// How to initialize plant control with helper methods in "FB_init()".
// [Hint]
// > All reference-variables are implemented to ease monitoring of relevant variables.
FUNCTION_BLOCK FB_Plt_Init2 EXTENDS FB_BA_View
VAR
   	{region 'Aggregates'}
		DmprSu_Open							: REFERENCE TO BOOL							REF= DmprSu.bOpen;
		DmprSu_Val							: REFERENCE TO REAL							REF= DmprSu.fActiveVal;
		DmprSu								: FB_TimerAggregateA						:= (iParent:=THIS^,					iLabel:=MyLabels.DmprSu);
		FanSu_Val							: REFERENCE TO UDINT						REF= FanSu.nActiveVal;
		FanSu								: FB_BA_AggregateM							:= (iParent:=THIS^,					iLabel:=MyLabels.FanSu);
			 
		DmprEx_Open							: REFERENCE TO BOOL							REF= DmprEx.bOpen;
		DmprEx_Val							: REFERENCE TO REAL							REF= DmprEx.fActiveVal;
		DmprEx								: FB_TimerAggregateA						:= (iParent:=THIS^,					iLabel:=MyLabels.DmprEx);
		FanEx_Val							: REFERENCE TO UDINT						REF= FanEx.nActiveVal;
		FanEx								: FB_BA_AggregateM							:= (iParent:=THIS^,					iLabel:=MyLabels.FanEx);
			 
		PreHtr_Proc							: REFERENCE TO BOOL							REF= PreHtr.Process.bActive;
		PreHtr_Val							: REFERENCE TO BOOL							REF= PreHtr.bActiveVal;
		PreHtr								: FB_ProcAggregateB							:= (iParent:=THIS^,					iLabel:=MyLabels.PreHtr,			Process:=(iLabel:=MyLabels.ProcPreRinse));
		Erc_Val								: REFERENCE TO BOOL							REF= Erc.bActiveVal;
		Erc									: FB_BA_AggregateB							:= (iParent:=THIS^,					iLabel:=MyLabels.Erc);
		Col_Val								: REFERENCE TO BOOL							REF= Col.bActiveVal;
		Col									: FB_BA_AggregateB							:= (iParent:=THIS^,					iLabel:=MyLabels.Col);
	{endregion}
	{region 'Plant'} 
		OpMode								: E_OpMod_AC								:= E_OpMod_AC.eOff;
		PlantCtrl_OpSta						: REFERENCE TO BOOL							REF= PlantCtrl.bOpSta;
		PlantCtrl_On						: REFERENCE TO BOOL							REF= PlantCtrl.bOn;
		PlantCtrl_PrVal						: REFERENCE TO UDINT						REF= PlantCtrl.nPresentValue;
		PlantCtrl_Step						: REFERENCE TO STRING						REF= PlantCtrl.sStep;
		PlantCtrl							: FB_BA_PlantCtrl							:= (iParent:=THIS^,					iLabel:=MyLabels.PltCtrl);
	{endregion}
END_VAR

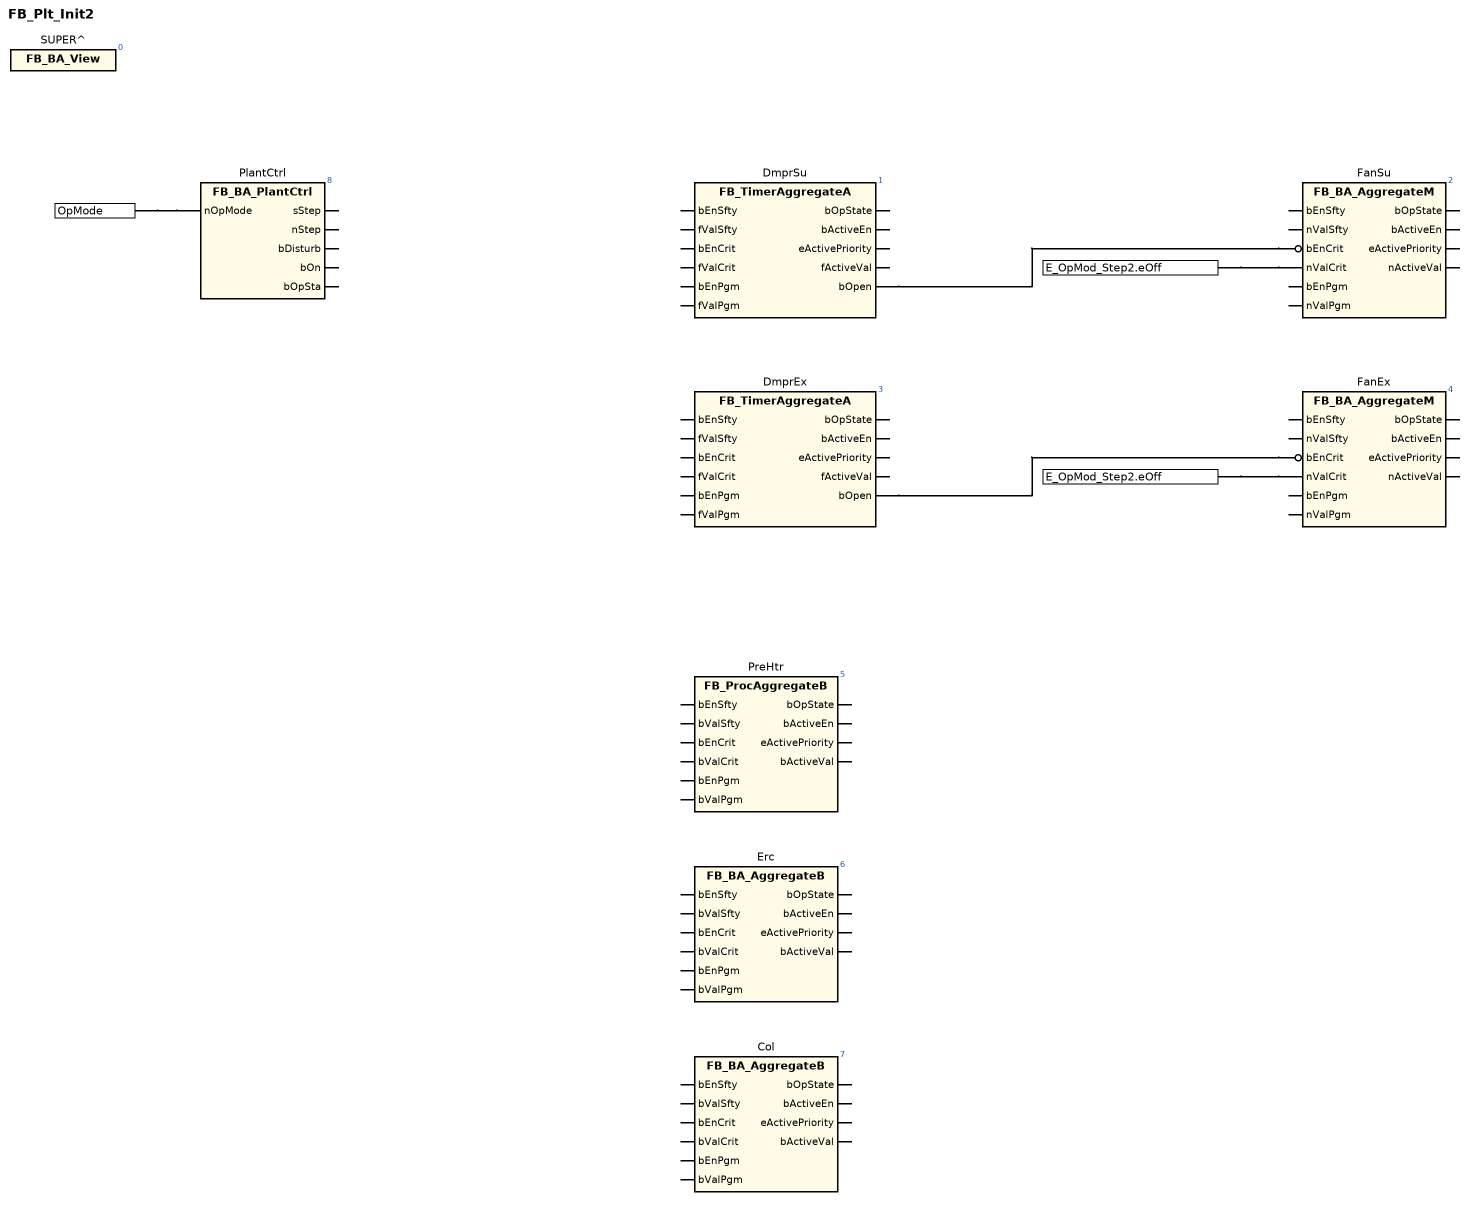
SUPER^(); // FB_BA_View
DmprSu(); // FB_TimerAggregateA
FanSu(bEnCrit := NOT DmprSu.bOpen, nValCrit := E_OpMod_Step2.eOff); // FB_BA_AggregateM
DmprEx(); // FB_TimerAggregateA
FanEx(bEnCrit := NOT DmprEx.bOpen, nValCrit := E_OpMod_Step2.eOff); // FB_BA_AggregateM
PreHtr(); // FB_ProcAggregateB
Erc(); // FB_BA_AggregateB
Col(); // FB_BA_AggregateB
PlantCtrl(nOpMode := OpMode); // FB_BA_PlantCtrl

METHOD FB_init : BOOL
VAR_INPUT
	bInitRetains : BOOL; // if TRUE, the retain variables are initialized (warm start / cold start)
	bInCopyCode : BOOL;  // if TRUE, the instance afterwards gets moved into the copy code (online change)
END_VAR
PlantCtrl.Clear();

// Add plant operations modes:
PlantCtrl.AddOperationMode(E_OpMod_AC.eDisturb,			E_BA_Priority.eCritical,	E_BA_AggregateIgnoreFlags.Delay);
PlantCtrl.AddOperationMode(E_OpMod_AC.eSmokeExtract,	E_BA_Priority.eLifeSafety,	E_BA_AggregateIgnoreFlags.All);
PlantCtrl.AddOperationMode(E_OpMod_AC.eOff,				E_BA_Priority.eProgram,		E_BA_AggregateIgnoreFlags.None);
PlantCtrl.AddOperationMode(E_OpMod_AC.eOn,				E_BA_Priority.eProgram,		E_BA_AggregateIgnoreFlags.None);
PlantCtrl.AddOperationMode(E_OpMod_AC.eNightCool,		E_BA_Priority.eProgram,		E_BA_AggregateIgnoreFlags.None);

// Add aggregates:
PlantCtrl.AddAggregate(DmprSu,	FALSE,	FALSE,	T#0S,	T#0S);
PlantCtrl.AddAggregate(DmprEx,	FALSE,	FALSE,	T#0S,	T#0S);
PlantCtrl.AddAggregate(PreHtr,	TRUE,	FALSE,	T#0S,	T#0S);
PlantCtrl.AddAggregate(Erc,		FALSE,	FALSE,	T#0S,	T#0S);
PlantCtrl.AddAggregate(Col,		FALSE,	FALSE,	T#0S,	T#0S);
PlantCtrl.AddAggregate(FanSu,	FALSE,	FALSE,	T#0S,	T#5S);
PlantCtrl.AddAggregate(FanEx,	FALSE,	FALSE,	T#5S,	T#0S);

// Apply aggregate operation modes dependant on corresponding plant operation modes:
PlantCtrl.AssignAggregate4x(E_OpMod_AC.eDisturb,		DmprSu, TO_UDINT(0),					FanSu, TO_UDINT(E_OpMod_Step2.eOff),		DmprEx, TO_UDINT(0),					FanEx, TO_UDINT(E_OpMod_Step2.eOff));
PlantCtrl.AssignAggregate4x(E_OpMod_AC.eSmokeExtract,	DmprSu, TO_UDINT(100),					FanSu, TO_UDINT(E_OpMod_Step2.eStep2),		DmprEx, TO_UDINT(100),					FanEx, TO_UDINT(E_OpMod_Step2.eStep2));
PlantCtrl.AssignAggregate4x(E_OpMod_AC.eOff,			DmprSu, TO_UDINT(0),					FanSu, TO_UDINT(E_OpMod_Step2.eOff),		DmprEx, TO_UDINT(0),					FanEx, TO_UDINT(E_OpMod_Step2.eOff));
PlantCtrl.AssignAggregate4x(E_OpMod_AC.eOn,				DmprSu, TO_UDINT(100),					FanSu, TO_UDINT(E_OpMod_Step2.eStep1),		DmprEx, TO_UDINT(100),					FanEx, TO_UDINT(E_OpMod_Step2.eStep1));
PlantCtrl.AssignAggregate4x(E_OpMod_AC.eNightCool,		DmprSu, TO_UDINT(100),					FanSu, TO_UDINT(E_OpMod_Step2.eStep2),		DmprEx, TO_UDINT(100),					FanEx, TO_UDINT(E_OpMod_Step2.eStep2));

PlantCtrl.AssignAggregate3x(E_OpMod_AC.eDisturb,		PreHtr, TO_UDINT(E_OpMod_Binary.eOff),	Erc, TO_UDINT(E_OpMod_Binary.eOff),			Col, TO_UDINT(E_OpMod_Binary.eOff));
PlantCtrl.AssignAggregate3x(E_OpMod_AC.eSmokeExtract,	PreHtr, TO_UDINT(E_OpMod_Binary.eOn),	Erc, TO_UDINT(E_OpMod_Binary.eOn),			Col, TO_UDINT(E_OpMod_Binary.eOn));
PlantCtrl.AssignAggregate3x(E_OpMod_AC.eOff,			PreHtr, TO_UDINT(E_OpMod_Binary.eOff),	Erc, TO_UDINT(E_OpMod_Binary.eOff),			Col, TO_UDINT(E_OpMod_Binary.eOff));
PlantCtrl.AssignAggregate3x(E_OpMod_AC.eOn,				PreHtr, TO_UDINT(E_OpMod_Binary.eOn),	Erc, TO_UDINT(E_OpMod_Binary.eOn),			Col, TO_UDINT(E_OpMod_Binary.eOn));
PlantCtrl.AssignAggregate3x(E_OpMod_AC.eNightCool,		PreHtr, TO_UDINT(E_OpMod_Binary.eOff),	Erc, TO_UDINT(E_OpMod_Binary.eOff),			Col, TO_UDINT(E_OpMod_Binary.eOff));
END_METHOD

END_FUNCTION_BLOCK

(* stored: Version 1.1.0.1, ProductVersion 3.1.4024.9
   POU FB_Plt_Init2: Id {ff8ee360-1381-48c8-ac76-513f54c50d79}, SpecialFunc None
   Method FB_init: Id {9ab58b83-86a7-4a29-afb5-e4bd42ff20de} *)
